// TwinCAT 3 PLC project New folder
// ProgramVersion: 3.1.4024.0
// libraries:
//   Tc2_Standard, * (Beckhoff Automation GmbH)
//   Tc2_System, * (Beckhoff Automation GmbH)
//   Tc3_Module, * (Beckhoff Automation GmbH)
// project tree:
//   GVLs/ GVL_ADS.TcGVL
//   / PlcTask.TcTTO
//   POUs/ MAIN.TcPOU

CONFIGURATION New_folder
    RESOURCE PLC ON TwinCAT3
        TASK PlcTask(INTERVAL := T#10ms, PRIORITY := 20);
        PROGRAM MAIN WITH PlcTask : MAIN;
    END_RESOURCE
END_CONFIGURATION

// ---- GVLs/GVL_ADS.TcGVL
{attribute 'Tc2GvlVarNames'}
VAR_GLOBAL
	Array_EPB_TDA_INT AT%MB1100:ARRAY [0..20] OF INT;
END_VAR

// ---- POUs/MAIN.TcPOU
PROGRAM MAIN
VAR
	i: INT;
END_VAR

FOR i := 0 TO 20 DO
	GVL_ADS.Array_EPB_TDA_INT[i] := i;
END_FOR

END_PROGRAM
